FUNCTION_BLOCK CAMERA_CAPTURE
  {SET_ATTRIBUTE(OpcUa, DEVICE.SENSOR)}
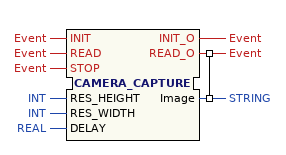
  EVENT_INPUT
    INIT;
    READ;
    STOP;
  END_EVENT
  EVENT_OUTPUT
    INIT_O;
    READ_O WITH Image;
  END_EVENT
  VAR_INPUT
    RES_HEIGHT : INT; (* Image height resolution *)
    RES_WIDTH : INT; (* Image width resolution *)
    DELAY : REAL; (* Delay before capturing (seconds) *)
  END_VAR
  VAR_OUTPUT
    Image : STRING;
  END_VAR
END_FUNCTION_BLOCK
